Staubli VAL3: ClientGet.pgx

public program ClientGet(string& x_sRes)
  local num l_nNum[200]
  local num l_nIndex
begin
  x_sRes=""

  //从服务器获得字符串
  if sioGet(sClient,l_nNum)<0
    return
  endIf

  wait(sioGet(sClient,l_nNum)>=0)

  //把Acsii转换为字符串
  for l_nIndex=0 to size(l_nNum)-1
    x_sRes=x_sRes+chr(l_nNum[l_nIndex])
  endFor

  //  wait((x_sRes=sClient)!="")

end
